# EPICS substitutions: ipmiMgrApp/Db/power_module.substitutions
#
# PM : Power Module Wiener AC1000
#          This is the standard PM for 9U MTCA crates
#
#
# nat> show_sensorinfo 51
# Sensor Information for FRU 51 / PM2
# ==================================================================
#   #   SDRType  Sensor Entity Inst  Value   State    Name
# ------------------------------------------------------------------
#   -   MDevLoc          0x0a  0x62                    PM-AC1000
#   1   Full     Temp    0x0a  0x62  36 C       ok     T DCDC UPD
#   2   Full     Temp    0x0a  0x62  34 C       ok     T PATH UPD
#   3   Full     Temp    0x0a  0x62  41 C       ok     T COOLER UPM
#   4   Full     Temp    0x0a  0x62  37 C       ok     T TRAFO UPM
#   5   Full     Voltage 0x0a  0x62  3.24 V     ok     MP
#   6   Full     Voltage 0x0a  0x62  4.98 V     ok     SMP
#   7   Full     Voltage 0x0a  0x62  4.98 V     ok     SMPP
#   8   Full     Voltage 0x0a  0x62  12.36 V    ok     PP
#   9   Full     Voltage 0x0a  0x62  11.40 V    ok     12VHH
#  10   Full     Current 0x0a  0x62  10.40 A    ok     Current(Sum)
#  11   Full     Current 0x0a  0x62  1.45 A     ok     Ch01 Current
#  12   Full     Current 0x0a  0x62  0.00 A     ok     Ch02 Current
#  13   Full     Current 0x0a  0x62  1.75 A     ok     Ch03 Current
#  14   Full     Current 0x0a  0x62  1.90 A     ok     Ch04 Current
#  15   Full     Current 0x0a  0x62  1.80 A     ok     Ch05 Current
#  16   Full     Current 0x0a  0x62  0.55 A     ok     Ch06 Current
#  17   Full     Current 0x0a  0x62  0.00 A     ok     Ch07 Current
#  18   Full     Current 0x0a  0x62  1.95 A     ok     Ch08 Current
#  19   Full     Current 0x0a  0x62  0.00 A     ok     Ch09 Current
#  20   Full     Current 0x0a  0x62  0.00 A     ok     Ch10 Current
#  21   Full     Current 0x0a  0x62  0.00 A     ok     Ch11 Current
#  22   Full     Current 0x0a  0x62  1.25 A     ok     Ch12 Current
#  23   Full     Current 0x0a  0x62  0.00 A     ok     Ch13 Current
#  24   Full     Current 0x0a  0x62  0.00 A     ok     Ch14 Current
#  25   Full     Current 0x0a  0x62  0.00 A     ok     Ch15 Current
#  26   Full     Current 0x0a  0x62  0.00 A     ok     Ch16 Current
#  27   Compact  0xf2    0x0a  0x62  0x01              HotSwap
#  28   Event       -    0x0a  0x00                    PwrChan
#  29   Event       -    0x0a  0x00                    PM_Stat
#  28   Compact  0xf0    0x0a  0x62  0x10              HS 051 PM2
# ------------------------------------------------------------------

file "fru_common.db"
{
   pattern { id		, fruid 	}
           { $(id)	, $(fruid)	}
}

file "sensor_ai.db"
{
    pattern { attr	, sensinst	, type	, fruid		, prefix }
            { TempCpu0	, 1		, 1	, $(fruid)	, $(id)  }
            { TempPath	, 2		, 1	, $(fruid)	, $(id)  }
            { TempCool	, 3		, 1	, $(fruid)	, $(id)  }
            { TempTraf	, 4		, 1	, $(fruid)	, $(id)  }
            { VoltMP00V	, 1		, 2	, $(fruid)	, $(id)  }
            { VoltSMP0V	, 2		, 2	, $(fruid)	, $(id)  }
            { VoltSMPPV	, 3		, 2	, $(fruid)	, $(id)  }
            { VoltPP00V	, 4		, 2	, $(fruid)	, $(id)  }
            { Volt12HHV	, 5		, 2	, $(fruid)	, $(id)  }
            { CurrSum	, 1		, 3	, $(fruid)	, $(id)  }
            { CurrCh01	, 2		, 3	, $(fruid)	, $(id)  }
            { CurrCh02	, 3		, 3	, $(fruid)	, $(id)  }
            { CurrCh03	, 4		, 3	, $(fruid)	, $(id)  }
            { CurrCh04	, 5		, 3	, $(fruid)	, $(id)  }
            { CurrCh05	, 6		, 3	, $(fruid)	, $(id)  }
            { CurrCh06	, 7		, 3	, $(fruid)	, $(id)  }
            { CurrCh07	, 8		, 3	, $(fruid)	, $(id)  }
            { CurrCh08	, 9		, 3	, $(fruid)	, $(id)  }
            { CurrCh09	, 10		, 3	, $(fruid)	, $(id)  }
            { CurrCh10	, 11		, 3	, $(fruid)	, $(id)  }
            { CurrCh11	, 12		, 3	, $(fruid)	, $(id)  }
            { CurrCh12	, 13		, 3	, $(fruid)	, $(id)  }
            { CurrCh13	, 14		, 3	, $(fruid)	, $(id)  }
            { CurrCh14	, 15		, 3	, $(fruid)	, $(id)  }
            { CurrCh15	, 16		, 3	, $(fruid)	, $(id)  }
            { CurrCh16	, 17		, 3	, $(fruid)	, $(id)  }
 }
